// TIA Portal V17 export
// export: Created 2023-03-03T06:58:18.2471944Z, ExportSetting WithDefaults, DisplayName Totally Integrated Automation Portal, DisplayVersion V17 Update 5, DisplayName TIA Portal Openness, DisplayVersion V17 Update 5, DisplayName TIA Portal Version Control Interface, DisplayVersion V17, DisplayName SINAMICS Startdrive Advanced, DisplayVersion V17 SP1, DisplayName SINAMICS DCC, DisplayVersion V17 Update 1, DisplayName SINAMICS Startdrive G130, G150, S120, S150, SINAMICS MV, S210, DisplayVersion V17 SP1, DisplayName SINAMICS Startdrive G110M, G120, G120C, G120D, G120P, G115D, DisplayVersion V17 SP1, DisplayName STEP 7 Professional, DisplayVersion V17 Update 5, DisplayName STEP 7 Safety, DisplayVersion V17, DisplayName WinCC Advanced, DisplayVersion V17 Update 5
FUNCTION "Start motor HYD unit" : Void   // FC700, LAD
TITLE = FC Gestione accensione motori centralina HYD
{ S7_Optimized_Access := 'FALSE' }
AUTHOR : Max
FAMILY : Taglio
NAME : FC_START_MOTORI_CENTRALINA_HYD
VERSION : 0.1
// stored: AutoNumber false, IsIECCheckEnabled false, SetENOAutomatically false, UDAEnableTagReadback false
   VAR_TEMP
      cmd_Star : Bool;
      cmd_Triangle : Bool;
      cmd_recycling : Bool;
   END_VAR
   VAR_TEMP   // added for the SCL form of the ladder/FBD networks
      _w1 : Bool;
   END_VAR
BEGIN

REGION Network 1: *************************** Avviamento motore ricircolo **********************************
END_REGION

REGION Network 2: Condizioni per abilitazione avviamento motore ricircolo centralina
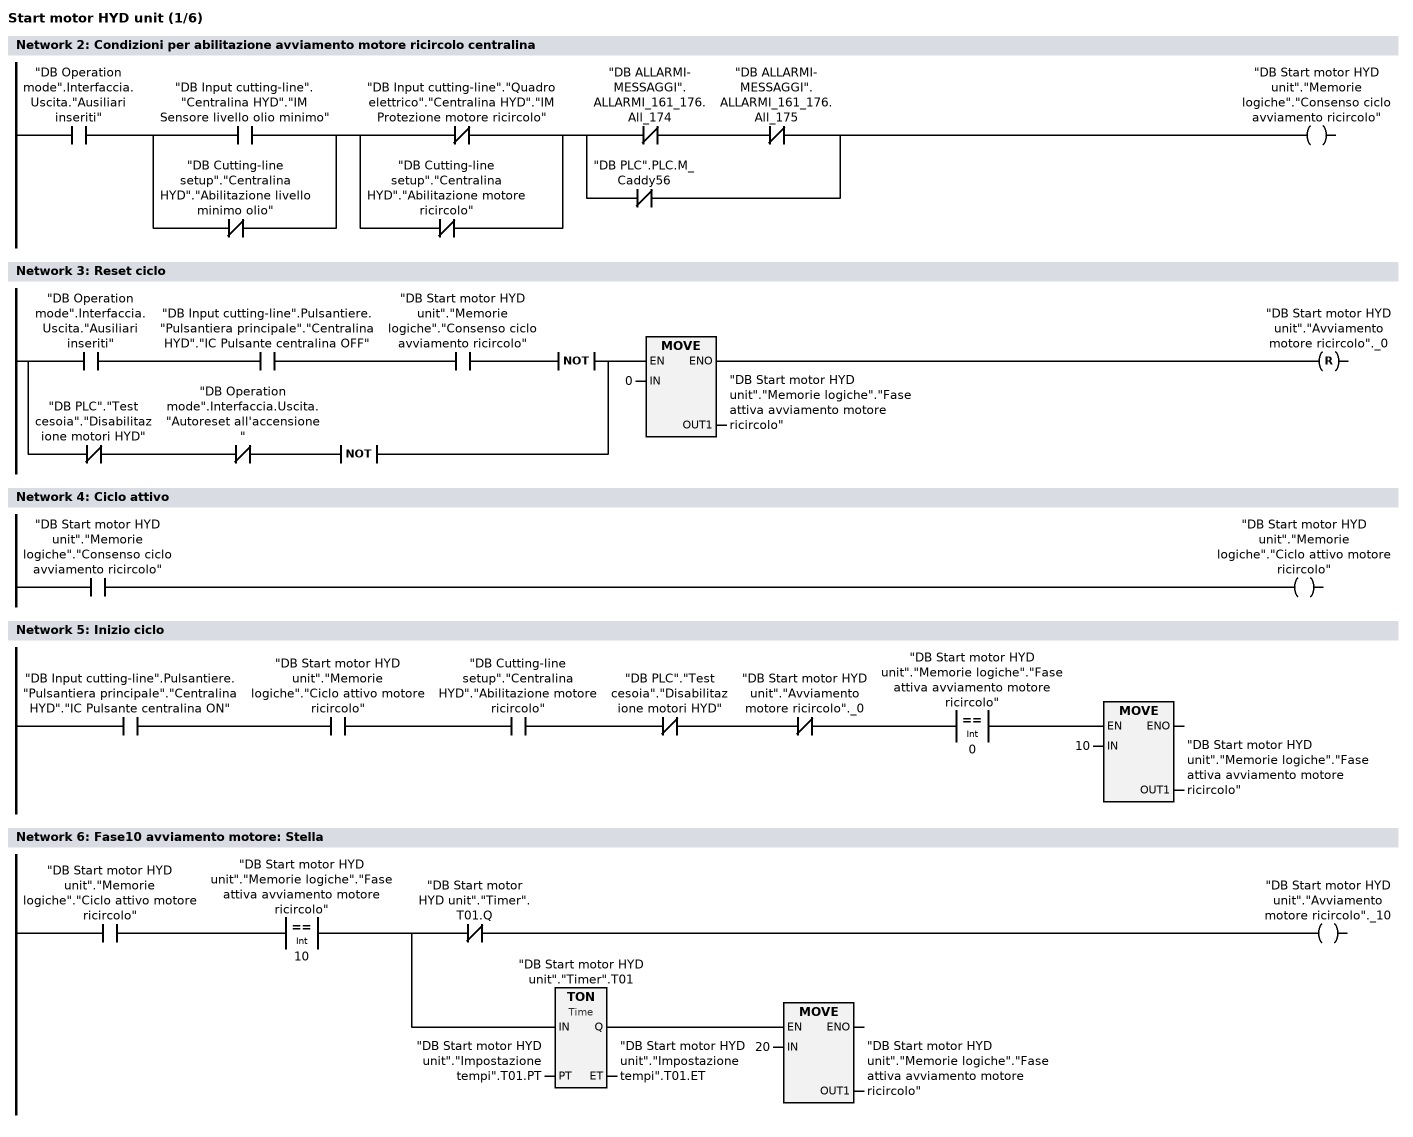
   RUNG wire#powerrail
      Contact( "DB Operation mode".Interfaccia.Uscita."Ausiliari inseriti" )
      wire#w1
      Contact( "DB Input cutting-line"."Centralina HYD"."IM Sensore livello olio minimo" )
      wire#w2
      I_Contact( "DB Input cutting-line"."Quadro elettrico"."Centralina HYD"."IM Protezione motore ricircolo" )
      wire#w3
      I_Contact( "DB ALLARMI-MESSAGGI".ALLARMI_161_176.All_174 )
      I_Contact( "DB ALLARMI-MESSAGGI".ALLARMI_161_176.All_175 )
      wire#w4
      Coil( "DB Start motor HYD unit"."Memorie logiche"."Consenso ciclo avviamento ricircolo" )
   END_RUNG
   RUNG wire#w1
      I_Contact( "DB Cutting-line setup"."Centralina HYD"."Abilitazione livello minimo olio" )
   END_RUNG wire#w2
   RUNG wire#w2
      I_Contact( "DB Cutting-line setup"."Centralina HYD"."Abilitazione motore ricircolo" )
   END_RUNG wire#w3
   RUNG wire#w3
      I_Contact( "DB PLC".PLC.M_Caddy56 )
   END_RUNG wire#w4
   // the same network as SCL:
   "DB Start motor HYD unit"."Memorie logiche"."Consenso ciclo avviamento ricircolo" := "DB Operation mode".Interfaccia.Uscita."Ausiliari inseriti" AND ("DB Input cutting-line"."Centralina HYD"."IM Sensore livello olio minimo" OR NOT "DB Cutting-line setup"."Centralina HYD"."Abilitazione livello minimo olio") AND (NOT "DB Input cutting-line"."Quadro elettrico"."Centralina HYD"."IM Protezione motore ricircolo" OR NOT "DB Cutting-line setup"."Centralina HYD"."Abilitazione motore ricircolo") AND ((NOT "DB ALLARMI-MESSAGGI".ALLARMI_161_176.All_174 AND NOT "DB ALLARMI-MESSAGGI".ALLARMI_161_176.All_175) OR NOT "DB PLC".PLC.M_Caddy56);
END_REGION

REGION Network 3: Reset ciclo
   RUNG wire#powerrail
      Contact( "DB Operation mode".Interfaccia.Uscita."Ausiliari inseriti" )
      Contact( "DB Input cutting-line".Pulsantiere."Pulsantiera principale"."Centralina HYD"."IC Pulsante centralina OFF" )
      Contact( "DB Start motor HYD unit"."Memorie logiche"."Consenso ciclo avviamento ricircolo" )
      Not()
      wire#w1
      Move(in := 0, out1 => "DB Start motor HYD unit"."Memorie logiche"."Fase attiva avviamento motore ricircolo")
      R_Coil( "DB Start motor HYD unit"."Avviamento motore ricircolo"._0 )
   END_RUNG
   RUNG wire#powerrail
      I_Contact( "DB PLC"."Test cesoia"."Disabilitazione motori HYD" )
      I_Contact( "DB Operation mode".Interfaccia.Uscita."Autoreset all'accensione" )
      Not()
   END_RUNG wire#w1
   // the same network as SCL:
   IF NOT ("DB Operation mode".Interfaccia.Uscita."Ausiliari inseriti" AND "DB Input cutting-line".Pulsantiere."Pulsantiera principale"."Centralina HYD"."IC Pulsante centralina OFF" AND "DB Start motor HYD unit"."Memorie logiche"."Consenso ciclo avviamento ricircolo") OR NOT (NOT "DB PLC"."Test cesoia"."Disabilitazione motori HYD" AND NOT "DB Operation mode".Interfaccia.Uscita."Autoreset all'accensione") THEN
       "DB Start motor HYD unit"."Memorie logiche"."Fase attiva avviamento motore ricircolo" := 0;
       "DB Start motor HYD unit"."Avviamento motore ricircolo"._0 := FALSE;
   END_IF;
END_REGION

REGION Network 4: Ciclo attivo
   RUNG wire#powerrail
      Contact( "DB Start motor HYD unit"."Memorie logiche"."Consenso ciclo avviamento ricircolo" )
      Coil( "DB Start motor HYD unit"."Memorie logiche"."Ciclo attivo motore ricircolo" )
   END_RUNG
   // the same network as SCL:
   "DB Start motor HYD unit"."Memorie logiche"."Ciclo attivo motore ricircolo" := "DB Start motor HYD unit"."Memorie logiche"."Consenso ciclo avviamento ricircolo";
END_REGION

REGION Network 5: Inizio ciclo
   RUNG wire#powerrail
      Contact( "DB Input cutting-line".Pulsantiere."Pulsantiera principale"."Centralina HYD"."IC Pulsante centralina ON" )
      Contact( "DB Start motor HYD unit"."Memorie logiche"."Ciclo attivo motore ricircolo" )
      Contact( "DB Cutting-line setup"."Centralina HYD"."Abilitazione motore ricircolo" )
      I_Contact( "DB PLC"."Test cesoia"."Disabilitazione motori HYD" )
      I_Contact( "DB Start motor HYD unit"."Avviamento motore ricircolo"._0 )
      { S7_Templates := "SrcType := Int" } EQ_Contact(in1 := "DB Start motor HYD unit"."Memorie logiche"."Fase attiva avviamento motore ricircolo", in2 := 0)
      Move(in := 10, out1 => "DB Start motor HYD unit"."Memorie logiche"."Fase attiva avviamento motore ricircolo")
   END_RUNG
   // the same network as SCL:
   IF "DB Input cutting-line".Pulsantiere."Pulsantiera principale"."Centralina HYD"."IC Pulsante centralina ON" AND "DB Start motor HYD unit"."Memorie logiche"."Ciclo attivo motore ricircolo" AND "DB Cutting-line setup"."Centralina HYD"."Abilitazione motore ricircolo" AND NOT "DB PLC"."Test cesoia"."Disabilitazione motori HYD" AND NOT "DB Start motor HYD unit"."Avviamento motore ricircolo"._0 AND ("DB Start motor HYD unit"."Memorie logiche"."Fase attiva avviamento motore ricircolo" = 0) THEN
       "DB Start motor HYD unit"."Memorie logiche"."Fase attiva avviamento motore ricircolo" := 10;
   END_IF;
END_REGION

REGION Network 6: Fase10 avviamento motore: Stella
   RUNG wire#powerrail
      Contact( "DB Start motor HYD unit"."Memorie logiche"."Ciclo attivo motore ricircolo" )
      { S7_Templates := "SrcType := Int" } EQ_Contact(in1 := "DB Start motor HYD unit"."Memorie logiche"."Fase attiva avviamento motore ricircolo", in2 := 10)
      wire#w1
      I_Contact( "DB Start motor HYD unit"."Timer".T01.Q )
      Coil( "DB Start motor HYD unit"."Avviamento motore ricircolo"._10 )
   END_RUNG
   RUNG wire#w1
      { S7_Templates := "time_type := Time" } "DB Start motor HYD unit"."Timer".T01.TON(pt := "DB Start motor HYD unit"."Impostazione tempi".T01.PT, et => "DB Start motor HYD unit"."Impostazione tempi".T01.ET)
      Move(in := 20, out1 => "DB Start motor HYD unit"."Memorie logiche"."Fase attiva avviamento motore ricircolo")
   END_RUNG
   // the same network as SCL:
   #_w1 := "DB Start motor HYD unit"."Memorie logiche"."Ciclo attivo motore ricircolo" AND ("DB Start motor HYD unit"."Memorie logiche"."Fase attiva avviamento motore ricircolo" = 10);
   "DB Start motor HYD unit"."Avviamento motore ricircolo"._10 := #_w1 AND NOT "DB Start motor HYD unit"."Timer".T01.Q;
   "DB Start motor HYD unit"."Timer".T01.TON(IN := #_w1,
                           PT := "DB Start motor HYD unit"."Impostazione tempi".T01.PT,
                           ET => "DB Start motor HYD unit"."Impostazione tempi".T01.ET);
   IF "DB Start motor HYD unit"."Timer".T01.Q THEN
       "DB Start motor HYD unit"."Memorie logiche"."Fase attiva avviamento motore ricircolo" := 20;
   END_IF;
END_REGION

REGION Network 7: Fase20 avviamento motore: Triangolo
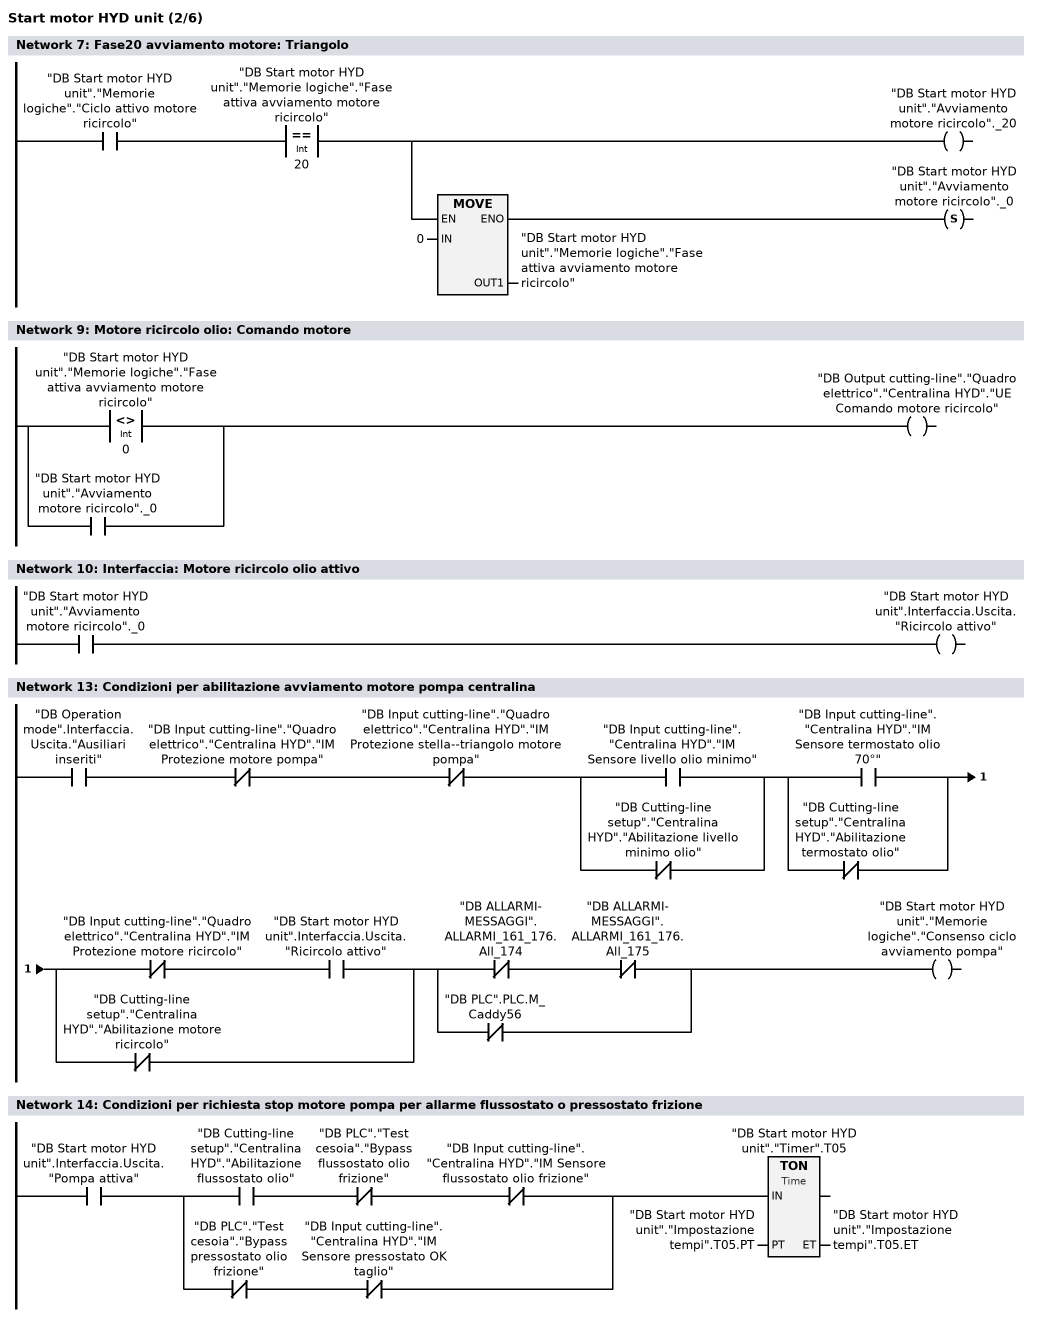
   RUNG wire#powerrail
      Contact( "DB Start motor HYD unit"."Memorie logiche"."Ciclo attivo motore ricircolo" )
      { S7_Templates := "SrcType := Int" } EQ_Contact(in1 := "DB Start motor HYD unit"."Memorie logiche"."Fase attiva avviamento motore ricircolo", in2 := 20)
      wire#w1
      Coil( "DB Start motor HYD unit"."Avviamento motore ricircolo"._20 )
   END_RUNG
   RUNG wire#w1
      Move(in := 0, out1 => "DB Start motor HYD unit"."Memorie logiche"."Fase attiva avviamento motore ricircolo")
      S_Coil( "DB Start motor HYD unit"."Avviamento motore ricircolo"._0 )
   END_RUNG
   // the same network as SCL:
   "DB Start motor HYD unit"."Avviamento motore ricircolo"._20 := "DB Start motor HYD unit"."Memorie logiche"."Ciclo attivo motore ricircolo" AND ("DB Start motor HYD unit"."Memorie logiche"."Fase attiva avviamento motore ricircolo" = 20);
   IF "DB Start motor HYD unit"."Avviamento motore ricircolo"._20 THEN
       "DB Start motor HYD unit"."Memorie logiche"."Fase attiva avviamento motore ricircolo" := 0;
       "DB Start motor HYD unit"."Avviamento motore ricircolo"._0 := TRUE;
   END_IF;
END_REGION

REGION Network 8: Dummy
END_REGION

REGION Network 9: Motore ricircolo olio: Comando motore
   RUNG wire#powerrail
      { S7_Templates := "SrcType := Int" } NE_Contact(in1 := "DB Start motor HYD unit"."Memorie logiche"."Fase attiva avviamento motore ricircolo", in2 := 0)
      wire#w1
      Coil( "DB Output cutting-line"."Quadro elettrico"."Centralina HYD"."UE Comando motore ricircolo" )
   END_RUNG
   RUNG wire#powerrail
      Contact( "DB Start motor HYD unit"."Avviamento motore ricircolo"._0 )
   END_RUNG wire#w1
   // the same network as SCL:
   "DB Output cutting-line"."Quadro elettrico"."Centralina HYD"."UE Comando motore ricircolo" := ("DB Start motor HYD unit"."Memorie logiche"."Fase attiva avviamento motore ricircolo" <> 0) OR "DB Start motor HYD unit"."Avviamento motore ricircolo"._0;
END_REGION

REGION Network 10: Interfaccia: Motore ricircolo olio attivo
   RUNG wire#powerrail
      Contact( "DB Start motor HYD unit"."Avviamento motore ricircolo"._0 )
      Coil( "DB Start motor HYD unit".Interfaccia.Uscita."Ricircolo attivo" )
   END_RUNG
   // the same network as SCL:
   "DB Start motor HYD unit".Interfaccia.Uscita."Ricircolo attivo" := "DB Start motor HYD unit"."Avviamento motore ricircolo"._0;
END_REGION

REGION Network 11: Dummy
END_REGION

REGION Network 12: *********************** Avviamento motore pompa principale ******************************
END_REGION

REGION Network 13: Condizioni per abilitazione avviamento motore pompa centralina
   RUNG wire#powerrail
      Contact( "DB Operation mode".Interfaccia.Uscita."Ausiliari inseriti" )
      I_Contact( "DB Input cutting-line"."Quadro elettrico"."Centralina HYD"."IM Protezione motore pompa" )
      I_Contact( "DB Input cutting-line"."Quadro elettrico"."Centralina HYD"."IM Protezione stella--triangolo motore pompa" )
      wire#w1
      Contact( "DB Input cutting-line"."Centralina HYD"."IM Sensore livello olio minimo" )
      wire#w2
      Contact( "DB Input cutting-line"."Centralina HYD"."IM Sensore termostato olio 70°" )
      wire#w3
      I_Contact( "DB Input cutting-line"."Quadro elettrico"."Centralina HYD"."IM Protezione motore ricircolo" )
      Contact( "DB Start motor HYD unit".Interfaccia.Uscita."Ricircolo attivo" )
      wire#w4
      I_Contact( "DB ALLARMI-MESSAGGI".ALLARMI_161_176.All_174 )
      I_Contact( "DB ALLARMI-MESSAGGI".ALLARMI_161_176.All_175 )
      wire#w5
      Coil( "DB Start motor HYD unit"."Memorie logiche"."Consenso ciclo avviamento pompa" )
   END_RUNG
   RUNG wire#w1
      I_Contact( "DB Cutting-line setup"."Centralina HYD"."Abilitazione livello minimo olio" )
   END_RUNG wire#w2
   RUNG wire#w2
      I_Contact( "DB Cutting-line setup"."Centralina HYD"."Abilitazione termostato olio" )
   END_RUNG wire#w3
   RUNG wire#w3
      I_Contact( "DB Cutting-line setup"."Centralina HYD"."Abilitazione motore ricircolo" )
   END_RUNG wire#w4
   RUNG wire#w4
      I_Contact( "DB PLC".PLC.M_Caddy56 )
   END_RUNG wire#w5
   // the same network as SCL:
   "DB Start motor HYD unit"."Memorie logiche"."Consenso ciclo avviamento pompa" := "DB Operation mode".Interfaccia.Uscita."Ausiliari inseriti" AND NOT "DB Input cutting-line"."Quadro elettrico"."Centralina HYD"."IM Protezione motore pompa" AND NOT "DB Input cutting-line"."Quadro elettrico"."Centralina HYD"."IM Protezione stella--triangolo motore pompa" AND ("DB Input cutting-line"."Centralina HYD"."IM Sensore livello olio minimo" OR NOT "DB Cutting-line setup"."Centralina HYD"."Abilitazione livello minimo olio") AND ("DB Input cutting-line"."Centralina HYD"."IM Sensore termostato olio 70°" OR NOT "DB Cutting-line setup"."Centralina HYD"."Abilitazione termostato olio") AND ((NOT "DB Input cutting-line"."Quadro elettrico"."Centralina HYD"."IM Protezione motore ricircolo" AND "DB Start motor HYD unit".Interfaccia.Uscita."Ricircolo attivo") OR NOT "DB Cutting-line setup"."Centralina HYD"."Abilitazione motore ricircolo") AND ((NOT "DB ALLARMI-MESSAGGI".ALLARMI_161_176.All_174 AND NOT "DB ALLARMI-MESSAGGI".ALLARMI_161_176.All_175) OR NOT "DB PLC".PLC.M_Caddy56);
END_REGION

REGION Network 14: Condizioni per richiesta stop motore pompa per allarme flussostato o pressostato frizione
   RUNG wire#powerrail
      Contact( "DB Start motor HYD unit".Interfaccia.Uscita."Pompa attiva" )
      wire#w1
      Contact( "DB Cutting-line setup"."Centralina HYD"."Abilitazione flussostato olio" )
      I_Contact( "DB PLC"."Test cesoia"."Bypass flussostato olio frizione" )
      I_Contact( "DB Input cutting-line"."Centralina HYD"."IM Sensore flussostato olio frizione" )
      wire#w2
      { S7_Templates := "time_type := Time" } "DB Start motor HYD unit"."Timer".T05.TON(pt := "DB Start motor HYD unit"."Impostazione tempi".T05.PT, et => "DB Start motor HYD unit"."Impostazione tempi".T05.ET)
   END_RUNG
   RUNG wire#w1
      I_Contact( "DB PLC"."Test cesoia"."Bypass pressostato olio frizione" )
      I_Contact( "DB Input cutting-line"."Centralina HYD"."IM Sensore pressostato OK taglio" )
   END_RUNG wire#w2
   // the same network as SCL:
   "DB Start motor HYD unit"."Timer".T05.TON(IN := "DB Start motor HYD unit".Interfaccia.Uscita."Pompa attiva" AND (("DB Cutting-line setup"."Centralina HYD"."Abilitazione flussostato olio" AND NOT "DB PLC"."Test cesoia"."Bypass flussostato olio frizione" AND NOT "DB Input cutting-line"."Centralina HYD"."IM Sensore flussostato olio frizione") OR (NOT "DB PLC"."Test cesoia"."Bypass pressostato olio frizione" AND NOT "DB Input cutting-line"."Centralina HYD"."IM Sensore pressostato OK taglio")),
                           PT := "DB Start motor HYD unit"."Impostazione tempi".T05.PT,
                           ET => "DB Start motor HYD unit"."Impostazione tempi".T05.ET);
END_REGION

REGION Network 15: Richiesta stop motore pompa per allarmi
   // Nel caso in cui avvengano allarmi viene usata questa richiesta. Cmq allo spegnimento degli ausiliari la pompa viene fermata dalla memoria "Ausiliari inseriti"
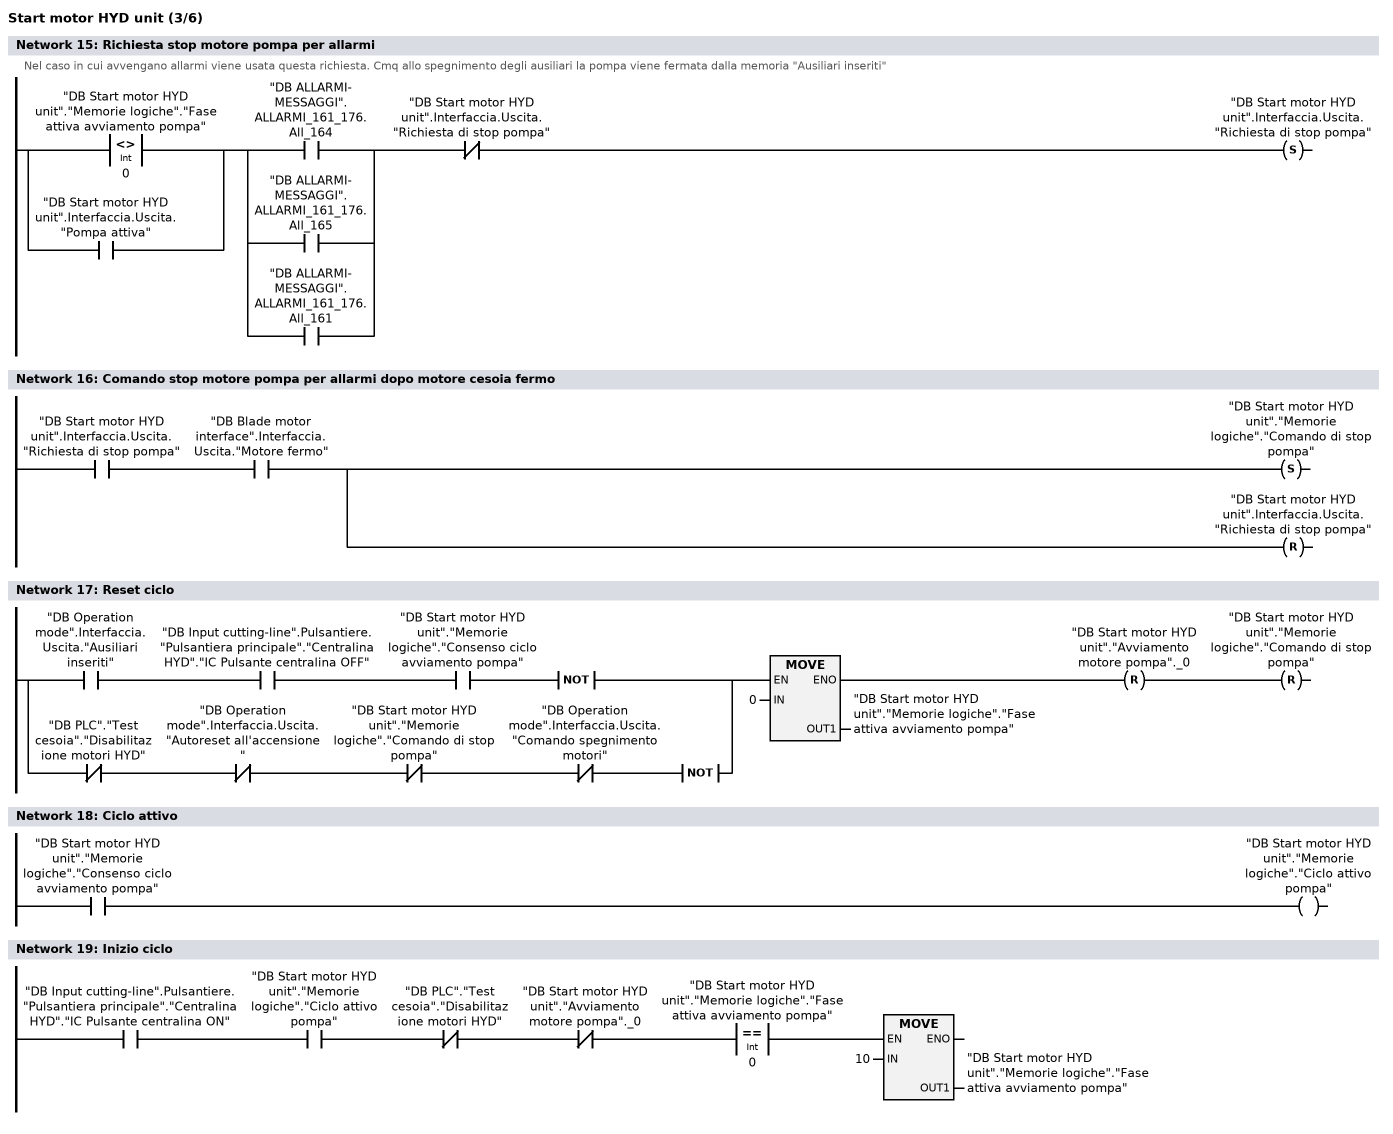
   RUNG wire#powerrail
      { S7_Templates := "SrcType := Int" } NE_Contact(in1 := "DB Start motor HYD unit"."Memorie logiche"."Fase attiva avviamento pompa", in2 := 0)
      wire#w1
      Contact( "DB ALLARMI-MESSAGGI".ALLARMI_161_176.All_164 )
      wire#w2
      I_Contact( "DB Start motor HYD unit".Interfaccia.Uscita."Richiesta di stop pompa" )
      S_Coil( "DB Start motor HYD unit".Interfaccia.Uscita."Richiesta di stop pompa" )
   END_RUNG
   RUNG wire#powerrail
      Contact( "DB Start motor HYD unit".Interfaccia.Uscita."Pompa attiva" )
   END_RUNG wire#w1
   RUNG wire#w1
      Contact( "DB ALLARMI-MESSAGGI".ALLARMI_161_176.All_165 )
   END_RUNG wire#w2
   RUNG wire#w1
      Contact( "DB ALLARMI-MESSAGGI".ALLARMI_161_176.All_161 )
   END_RUNG wire#w2
   // the same network as SCL:
   IF (("DB Start motor HYD unit"."Memorie logiche"."Fase attiva avviamento pompa" <> 0) OR "DB Start motor HYD unit".Interfaccia.Uscita."Pompa attiva") AND ("DB ALLARMI-MESSAGGI".ALLARMI_161_176.All_164 OR "DB ALLARMI-MESSAGGI".ALLARMI_161_176.All_165 OR "DB ALLARMI-MESSAGGI".ALLARMI_161_176.All_161) AND NOT "DB Start motor HYD unit".Interfaccia.Uscita."Richiesta di stop pompa" THEN
       "DB Start motor HYD unit".Interfaccia.Uscita."Richiesta di stop pompa" := TRUE;
   END_IF;
END_REGION

REGION Network 16: Comando stop motore pompa per allarmi dopo motore cesoia fermo
   RUNG wire#powerrail
      Contact( "DB Start motor HYD unit".Interfaccia.Uscita."Richiesta di stop pompa" )
      Contact( "DB Blade motor interface".Interfaccia.Uscita."Motore fermo" )
      wire#w1
      S_Coil( "DB Start motor HYD unit"."Memorie logiche"."Comando di stop pompa" )
   END_RUNG
   RUNG wire#w1
      R_Coil( "DB Start motor HYD unit".Interfaccia.Uscita."Richiesta di stop pompa" )
   END_RUNG
   // the same network as SCL:
   IF "DB Start motor HYD unit".Interfaccia.Uscita."Richiesta di stop pompa" AND "DB Blade motor interface".Interfaccia.Uscita."Motore fermo" THEN
       "DB Start motor HYD unit"."Memorie logiche"."Comando di stop pompa" := TRUE;
       "DB Start motor HYD unit".Interfaccia.Uscita."Richiesta di stop pompa" := FALSE;
   END_IF;
END_REGION

REGION Network 17: Reset ciclo
   RUNG wire#powerrail
      Contact( "DB Operation mode".Interfaccia.Uscita."Ausiliari inseriti" )
      Contact( "DB Input cutting-line".Pulsantiere."Pulsantiera principale"."Centralina HYD"."IC Pulsante centralina OFF" )
      Contact( "DB Start motor HYD unit"."Memorie logiche"."Consenso ciclo avviamento pompa" )
      Not()
      wire#w1
      Move(in := 0, out1 => "DB Start motor HYD unit"."Memorie logiche"."Fase attiva avviamento pompa")
      R_Coil( "DB Start motor HYD unit"."Avviamento motore pompa"._0 )
      R_Coil( "DB Start motor HYD unit"."Memorie logiche"."Comando di stop pompa" )
   END_RUNG
   RUNG wire#powerrail
      I_Contact( "DB PLC"."Test cesoia"."Disabilitazione motori HYD" )
      I_Contact( "DB Operation mode".Interfaccia.Uscita."Autoreset all'accensione" )
      I_Contact( "DB Start motor HYD unit"."Memorie logiche"."Comando di stop pompa" )
      I_Contact( "DB Operation mode".Interfaccia.Uscita."Comando spegnimento motori" )
      Not()
   END_RUNG wire#w1
   // the same network as SCL:
   IF NOT ("DB Operation mode".Interfaccia.Uscita."Ausiliari inseriti" AND "DB Input cutting-line".Pulsantiere."Pulsantiera principale"."Centralina HYD"."IC Pulsante centralina OFF" AND "DB Start motor HYD unit"."Memorie logiche"."Consenso ciclo avviamento pompa") OR NOT (NOT "DB PLC"."Test cesoia"."Disabilitazione motori HYD" AND NOT "DB Operation mode".Interfaccia.Uscita."Autoreset all'accensione" AND NOT "DB Start motor HYD unit"."Memorie logiche"."Comando di stop pompa" AND NOT "DB Operation mode".Interfaccia.Uscita."Comando spegnimento motori") THEN
       "DB Start motor HYD unit"."Memorie logiche"."Fase attiva avviamento pompa" := 0;
       "DB Start motor HYD unit"."Avviamento motore pompa"._0 := FALSE;
       "DB Start motor HYD unit"."Memorie logiche"."Comando di stop pompa" := FALSE;
   END_IF;
END_REGION

REGION Network 18: Ciclo attivo
   RUNG wire#powerrail
      Contact( "DB Start motor HYD unit"."Memorie logiche"."Consenso ciclo avviamento pompa" )
      Coil( "DB Start motor HYD unit"."Memorie logiche"."Ciclo attivo pompa" )
   END_RUNG
   // the same network as SCL:
   "DB Start motor HYD unit"."Memorie logiche"."Ciclo attivo pompa" := "DB Start motor HYD unit"."Memorie logiche"."Consenso ciclo avviamento pompa";
END_REGION

REGION Network 19: Inizio ciclo
   RUNG wire#powerrail
      Contact( "DB Input cutting-line".Pulsantiere."Pulsantiera principale"."Centralina HYD"."IC Pulsante centralina ON" )
      Contact( "DB Start motor HYD unit"."Memorie logiche"."Ciclo attivo pompa" )
      I_Contact( "DB PLC"."Test cesoia"."Disabilitazione motori HYD" )
      I_Contact( "DB Start motor HYD unit"."Avviamento motore pompa"._0 )
      { S7_Templates := "SrcType := Int" } EQ_Contact(in1 := "DB Start motor HYD unit"."Memorie logiche"."Fase attiva avviamento pompa", in2 := 0)
      Move(in := 10, out1 => "DB Start motor HYD unit"."Memorie logiche"."Fase attiva avviamento pompa")
   END_RUNG
   // the same network as SCL:
   IF "DB Input cutting-line".Pulsantiere."Pulsantiera principale"."Centralina HYD"."IC Pulsante centralina ON" AND "DB Start motor HYD unit"."Memorie logiche"."Ciclo attivo pompa" AND NOT "DB PLC"."Test cesoia"."Disabilitazione motori HYD" AND NOT "DB Start motor HYD unit"."Avviamento motore pompa"._0 AND ("DB Start motor HYD unit"."Memorie logiche"."Fase attiva avviamento pompa" = 0) THEN
       "DB Start motor HYD unit"."Memorie logiche"."Fase attiva avviamento pompa" := 10;
   END_IF;
END_REGION

REGION Network 20: Fase10 avviamento motore: Stella
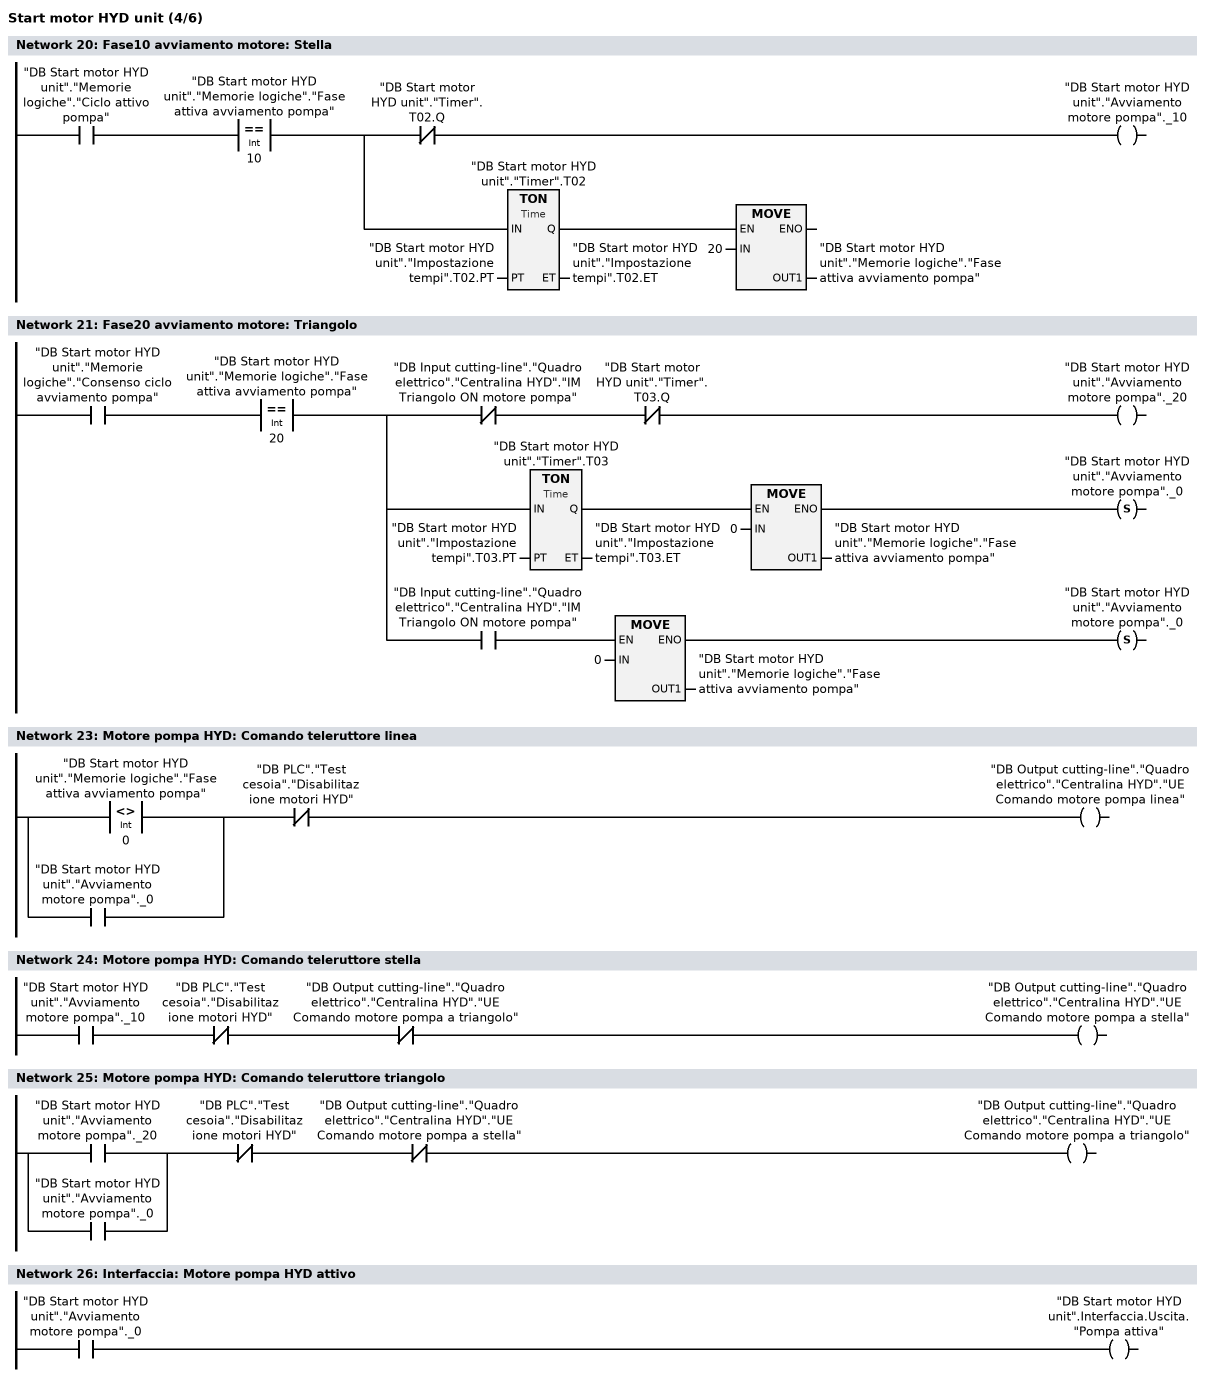
   RUNG wire#powerrail
      Contact( "DB Start motor HYD unit"."Memorie logiche"."Ciclo attivo pompa" )
      { S7_Templates := "SrcType := Int" } EQ_Contact(in1 := "DB Start motor HYD unit"."Memorie logiche"."Fase attiva avviamento pompa", in2 := 10)
      wire#w1
      I_Contact( "DB Start motor HYD unit"."Timer".T02.Q )
      Coil( "DB Start motor HYD unit"."Avviamento motore pompa"._10 )
   END_RUNG
   RUNG wire#w1
      { S7_Templates := "time_type := Time" } "DB Start motor HYD unit"."Timer".T02.TON(pt := "DB Start motor HYD unit"."Impostazione tempi".T02.PT, et => "DB Start motor HYD unit"."Impostazione tempi".T02.ET)
      Move(in := 20, out1 => "DB Start motor HYD unit"."Memorie logiche"."Fase attiva avviamento pompa")
   END_RUNG
   // the same network as SCL:
   #_w1 := "DB Start motor HYD unit"."Memorie logiche"."Ciclo attivo pompa" AND ("DB Start motor HYD unit"."Memorie logiche"."Fase attiva avviamento pompa" = 10);
   "DB Start motor HYD unit"."Avviamento motore pompa"._10 := #_w1 AND NOT "DB Start motor HYD unit"."Timer".T02.Q;
   "DB Start motor HYD unit"."Timer".T02.TON(IN := #_w1,
                           PT := "DB Start motor HYD unit"."Impostazione tempi".T02.PT,
                           ET => "DB Start motor HYD unit"."Impostazione tempi".T02.ET);
   IF "DB Start motor HYD unit"."Timer".T02.Q THEN
       "DB Start motor HYD unit"."Memorie logiche"."Fase attiva avviamento pompa" := 20;
   END_IF;
END_REGION

REGION Network 21: Fase20 avviamento motore: Triangolo
   RUNG wire#powerrail
      Contact( "DB Start motor HYD unit"."Memorie logiche"."Consenso ciclo avviamento pompa" )
      { S7_Templates := "SrcType := Int" } EQ_Contact(in1 := "DB Start motor HYD unit"."Memorie logiche"."Fase attiva avviamento pompa", in2 := 20)
      wire#w1
      I_Contact( "DB Input cutting-line"."Quadro elettrico"."Centralina HYD"."IM Triangolo ON motore pompa" )
      I_Contact( "DB Start motor HYD unit"."Timer".T03.Q )
      Coil( "DB Start motor HYD unit"."Avviamento motore pompa"._20 )
   END_RUNG
   RUNG wire#w1
      { S7_Templates := "time_type := Time" } "DB Start motor HYD unit"."Timer".T03.TON(pt := "DB Start motor HYD unit"."Impostazione tempi".T03.PT, et => "DB Start motor HYD unit"."Impostazione tempi".T03.ET)
      Move(in := 0, out1 => "DB Start motor HYD unit"."Memorie logiche"."Fase attiva avviamento pompa")
      S_Coil( "DB Start motor HYD unit"."Avviamento motore pompa"._0 )
   END_RUNG
   RUNG wire#w1
      Contact( "DB Input cutting-line"."Quadro elettrico"."Centralina HYD"."IM Triangolo ON motore pompa" )
      Move(in := 0, out1 => "DB Start motor HYD unit"."Memorie logiche"."Fase attiva avviamento pompa")
      S_Coil( "DB Start motor HYD unit"."Avviamento motore pompa"._0 )
   END_RUNG
   // the same network as SCL:
   #_w1 := "DB Start motor HYD unit"."Memorie logiche"."Consenso ciclo avviamento pompa" AND ("DB Start motor HYD unit"."Memorie logiche"."Fase attiva avviamento pompa" = 20);
   "DB Start motor HYD unit"."Avviamento motore pompa"._20 := #_w1 AND NOT "DB Input cutting-line"."Quadro elettrico"."Centralina HYD"."IM Triangolo ON motore pompa" AND NOT "DB Start motor HYD unit"."Timer".T03.Q;
   "DB Start motor HYD unit"."Timer".T03.TON(IN := #_w1,
                           PT := "DB Start motor HYD unit"."Impostazione tempi".T03.PT,
                           ET => "DB Start motor HYD unit"."Impostazione tempi".T03.ET);
   IF "DB Start motor HYD unit"."Timer".T03.Q THEN
       "DB Start motor HYD unit"."Memorie logiche"."Fase attiva avviamento pompa" := 0;
       "DB Start motor HYD unit"."Avviamento motore pompa"._0 := TRUE;
   END_IF;
   IF #_w1 AND "DB Input cutting-line"."Quadro elettrico"."Centralina HYD"."IM Triangolo ON motore pompa" THEN
       "DB Start motor HYD unit"."Memorie logiche"."Fase attiva avviamento pompa" := 0;
       "DB Start motor HYD unit"."Avviamento motore pompa"._0 := TRUE;
   END_IF;
END_REGION

REGION Network 22: Dummy
END_REGION

REGION Network 23: Motore pompa HYD: Comando teleruttore linea
   RUNG wire#powerrail
      { S7_Templates := "SrcType := Int" } NE_Contact(in1 := "DB Start motor HYD unit"."Memorie logiche"."Fase attiva avviamento pompa", in2 := 0)
      wire#w1
      I_Contact( "DB PLC"."Test cesoia"."Disabilitazione motori HYD" )
      Coil( "DB Output cutting-line"."Quadro elettrico"."Centralina HYD"."UE Comando motore pompa linea" )
   END_RUNG
   RUNG wire#powerrail
      Contact( "DB Start motor HYD unit"."Avviamento motore pompa"._0 )
   END_RUNG wire#w1
   // the same network as SCL:
   "DB Output cutting-line"."Quadro elettrico"."Centralina HYD"."UE Comando motore pompa linea" := (("DB Start motor HYD unit"."Memorie logiche"."Fase attiva avviamento pompa" <> 0) OR "DB Start motor HYD unit"."Avviamento motore pompa"._0) AND NOT "DB PLC"."Test cesoia"."Disabilitazione motori HYD";
END_REGION

REGION Network 24: Motore pompa HYD: Comando teleruttore stella
   RUNG wire#powerrail
      Contact( "DB Start motor HYD unit"."Avviamento motore pompa"._10 )
      I_Contact( "DB PLC"."Test cesoia"."Disabilitazione motori HYD" )
      I_Contact( "DB Output cutting-line"."Quadro elettrico"."Centralina HYD"."UE Comando motore pompa a triangolo" )
      Coil( "DB Output cutting-line"."Quadro elettrico"."Centralina HYD"."UE Comando motore pompa a stella" )
   END_RUNG
   // the same network as SCL:
   "DB Output cutting-line"."Quadro elettrico"."Centralina HYD"."UE Comando motore pompa a stella" := "DB Start motor HYD unit"."Avviamento motore pompa"._10 AND NOT "DB PLC"."Test cesoia"."Disabilitazione motori HYD" AND NOT "DB Output cutting-line"."Quadro elettrico"."Centralina HYD"."UE Comando motore pompa a triangolo";
END_REGION

REGION Network 25: Motore pompa HYD: Comando teleruttore triangolo
   RUNG wire#powerrail
      Contact( "DB Start motor HYD unit"."Avviamento motore pompa"._20 )
      wire#w1
      I_Contact( "DB PLC"."Test cesoia"."Disabilitazione motori HYD" )
      I_Contact( "DB Output cutting-line"."Quadro elettrico"."Centralina HYD"."UE Comando motore pompa a stella" )
      Coil( "DB Output cutting-line"."Quadro elettrico"."Centralina HYD"."UE Comando motore pompa a triangolo" )
   END_RUNG
   RUNG wire#powerrail
      Contact( "DB Start motor HYD unit"."Avviamento motore pompa"._0 )
   END_RUNG wire#w1
   // the same network as SCL:
   "DB Output cutting-line"."Quadro elettrico"."Centralina HYD"."UE Comando motore pompa a triangolo" := ("DB Start motor HYD unit"."Avviamento motore pompa"._20 OR "DB Start motor HYD unit"."Avviamento motore pompa"._0) AND NOT "DB PLC"."Test cesoia"."Disabilitazione motori HYD" AND NOT "DB Output cutting-line"."Quadro elettrico"."Centralina HYD"."UE Comando motore pompa a stella";
END_REGION

REGION Network 26: Interfaccia: Motore pompa HYD attivo
   RUNG wire#powerrail
      Contact( "DB Start motor HYD unit"."Avviamento motore pompa"._0 )
      Coil( "DB Start motor HYD unit".Interfaccia.Uscita."Pompa attiva" )
   END_RUNG
   // the same network as SCL:
   "DB Start motor HYD unit".Interfaccia.Uscita."Pompa attiva" := "DB Start motor HYD unit"."Avviamento motore pompa"._0;
END_REGION

REGION Network 27: Dummy
END_REGION

REGION Network 28: Comando valvola pressione olio cesoia
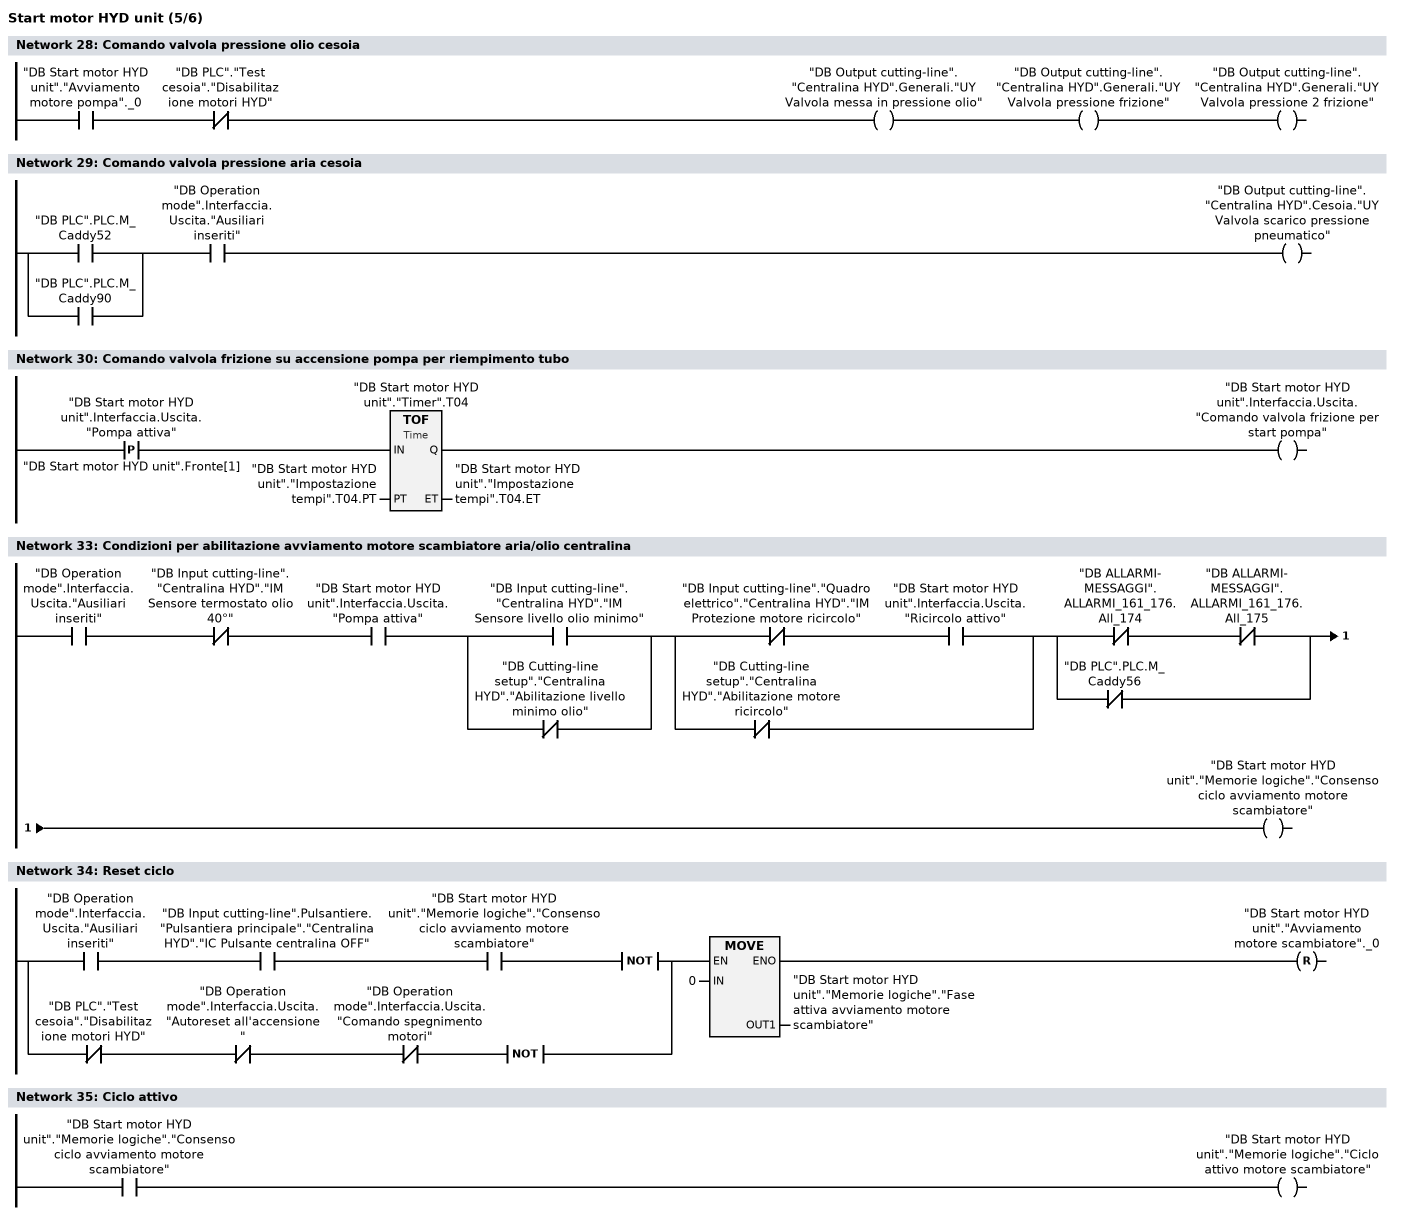
   RUNG wire#powerrail
      Contact( "DB Start motor HYD unit"."Avviamento motore pompa"._0 )
      I_Contact( "DB PLC"."Test cesoia"."Disabilitazione motori HYD" )
      Coil( "DB Output cutting-line"."Centralina HYD".Generali."UY Valvola messa in pressione olio" )
      Coil( "DB Output cutting-line"."Centralina HYD".Generali."UY Valvola pressione frizione" )
      Coil( "DB Output cutting-line"."Centralina HYD".Generali."UY Valvola pressione 2 frizione" )
   END_RUNG
   // the same network as SCL:
   "DB Output cutting-line"."Centralina HYD".Generali."UY Valvola messa in pressione olio" := "DB Start motor HYD unit"."Avviamento motore pompa"._0 AND NOT "DB PLC"."Test cesoia"."Disabilitazione motori HYD";
   "DB Output cutting-line"."Centralina HYD".Generali."UY Valvola pressione frizione" := "DB Output cutting-line"."Centralina HYD".Generali."UY Valvola messa in pressione olio";
   "DB Output cutting-line"."Centralina HYD".Generali."UY Valvola pressione 2 frizione" := "DB Output cutting-line"."Centralina HYD".Generali."UY Valvola messa in pressione olio";
END_REGION

REGION Network 29: Comando valvola pressione aria cesoia
   RUNG wire#powerrail
      Contact( "DB PLC".PLC.M_Caddy52 )
      wire#w1
      Contact( "DB Operation mode".Interfaccia.Uscita."Ausiliari inseriti" )
      Coil( "DB Output cutting-line"."Centralina HYD".Cesoia."UY Valvola scarico pressione pneumatico" )
   END_RUNG
   RUNG wire#powerrail
      Contact( "DB PLC".PLC.M_Caddy90 )
   END_RUNG wire#w1
   // the same network as SCL:
   "DB Output cutting-line"."Centralina HYD".Cesoia."UY Valvola scarico pressione pneumatico" := ("DB PLC".PLC.M_Caddy52 OR "DB PLC".PLC.M_Caddy90) AND "DB Operation mode".Interfaccia.Uscita."Ausiliari inseriti";
END_REGION

REGION Network 30: Comando valvola frizione su accensione pompa per riempimento tubo
   RUNG wire#powerrail
      P_Contact(operand := "DB Start motor HYD unit".Interfaccia.Uscita."Pompa attiva", bit := "DB Start motor HYD unit".Fronte[1])
      { S7_Templates := "time_type := Time" } "DB Start motor HYD unit"."Timer".T04.TOF(pt := "DB Start motor HYD unit"."Impostazione tempi".T04.PT, et => "DB Start motor HYD unit"."Impostazione tempi".T04.ET)
      Coil( "DB Start motor HYD unit".Interfaccia.Uscita."Comando valvola frizione per start pompa" )
   END_RUNG
   // the same network as SCL:
   #_w1 := "DB Start motor HYD unit".Interfaccia.Uscita."Pompa attiva" AND NOT "DB Start motor HYD unit".Fronte[1];   // rising edge of "DB Start motor HYD unit".Interfaccia.Uscita."Pompa attiva"
   "DB Start motor HYD unit".Fronte[1] := "DB Start motor HYD unit".Interfaccia.Uscita."Pompa attiva";
   "DB Start motor HYD unit"."Timer".T04.TOF(IN := #_w1,
                           PT := "DB Start motor HYD unit"."Impostazione tempi".T04.PT,
                           ET => "DB Start motor HYD unit"."Impostazione tempi".T04.ET);
   "DB Start motor HYD unit".Interfaccia.Uscita."Comando valvola frizione per start pompa" := "DB Start motor HYD unit"."Timer".T04.Q;
END_REGION

REGION Network 31: Dummy
END_REGION

REGION Network 32: *********************** Avviamento motore scambiatore aria/olio ****************************
END_REGION

REGION Network 33: Condizioni per abilitazione avviamento motore scambiatore aria/olio centralina
   RUNG wire#powerrail
      Contact( "DB Operation mode".Interfaccia.Uscita."Ausiliari inseriti" )
      I_Contact( "DB Input cutting-line"."Centralina HYD"."IM Sensore termostato olio 40°" )
      Contact( "DB Start motor HYD unit".Interfaccia.Uscita."Pompa attiva" )
      wire#w1
      Contact( "DB Input cutting-line"."Centralina HYD"."IM Sensore livello olio minimo" )
      wire#w2
      I_Contact( "DB Input cutting-line"."Quadro elettrico"."Centralina HYD"."IM Protezione motore ricircolo" )
      Contact( "DB Start motor HYD unit".Interfaccia.Uscita."Ricircolo attivo" )
      wire#w3
      I_Contact( "DB ALLARMI-MESSAGGI".ALLARMI_161_176.All_174 )
      I_Contact( "DB ALLARMI-MESSAGGI".ALLARMI_161_176.All_175 )
      wire#w4
      Coil( "DB Start motor HYD unit"."Memorie logiche"."Consenso ciclo avviamento motore scambiatore" )
   END_RUNG
   RUNG wire#w1
      I_Contact( "DB Cutting-line setup"."Centralina HYD"."Abilitazione livello minimo olio" )
   END_RUNG wire#w2
   RUNG wire#w2
      I_Contact( "DB Cutting-line setup"."Centralina HYD"."Abilitazione motore ricircolo" )
   END_RUNG wire#w3
   RUNG wire#w3
      I_Contact( "DB PLC".PLC.M_Caddy56 )
   END_RUNG wire#w4
   // the same network as SCL:
   "DB Start motor HYD unit"."Memorie logiche"."Consenso ciclo avviamento motore scambiatore" := "DB Operation mode".Interfaccia.Uscita."Ausiliari inseriti" AND NOT "DB Input cutting-line"."Centralina HYD"."IM Sensore termostato olio 40°" AND "DB Start motor HYD unit".Interfaccia.Uscita."Pompa attiva" AND ("DB Input cutting-line"."Centralina HYD"."IM Sensore livello olio minimo" OR NOT "DB Cutting-line setup"."Centralina HYD"."Abilitazione livello minimo olio") AND ((NOT "DB Input cutting-line"."Quadro elettrico"."Centralina HYD"."IM Protezione motore ricircolo" AND "DB Start motor HYD unit".Interfaccia.Uscita."Ricircolo attivo") OR NOT "DB Cutting-line setup"."Centralina HYD"."Abilitazione motore ricircolo") AND ((NOT "DB ALLARMI-MESSAGGI".ALLARMI_161_176.All_174 AND NOT "DB ALLARMI-MESSAGGI".ALLARMI_161_176.All_175) OR NOT "DB PLC".PLC.M_Caddy56);
END_REGION

REGION Network 34: Reset ciclo
   RUNG wire#powerrail
      Contact( "DB Operation mode".Interfaccia.Uscita."Ausiliari inseriti" )
      Contact( "DB Input cutting-line".Pulsantiere."Pulsantiera principale"."Centralina HYD"."IC Pulsante centralina OFF" )
      Contact( "DB Start motor HYD unit"."Memorie logiche"."Consenso ciclo avviamento motore scambiatore" )
      Not()
      wire#w1
      Move(in := 0, out1 => "DB Start motor HYD unit"."Memorie logiche"."Fase attiva avviamento motore scambiatore")
      R_Coil( "DB Start motor HYD unit"."Avviamento motore scambiatore"._0 )
   END_RUNG
   RUNG wire#powerrail
      I_Contact( "DB PLC"."Test cesoia"."Disabilitazione motori HYD" )
      I_Contact( "DB Operation mode".Interfaccia.Uscita."Autoreset all'accensione" )
      I_Contact( "DB Operation mode".Interfaccia.Uscita."Comando spegnimento motori" )
      Not()
   END_RUNG wire#w1
   // the same network as SCL:
   IF NOT ("DB Operation mode".Interfaccia.Uscita."Ausiliari inseriti" AND "DB Input cutting-line".Pulsantiere."Pulsantiera principale"."Centralina HYD"."IC Pulsante centralina OFF" AND "DB Start motor HYD unit"."Memorie logiche"."Consenso ciclo avviamento motore scambiatore") OR NOT (NOT "DB PLC"."Test cesoia"."Disabilitazione motori HYD" AND NOT "DB Operation mode".Interfaccia.Uscita."Autoreset all'accensione" AND NOT "DB Operation mode".Interfaccia.Uscita."Comando spegnimento motori") THEN
       "DB Start motor HYD unit"."Memorie logiche"."Fase attiva avviamento motore scambiatore" := 0;
       "DB Start motor HYD unit"."Avviamento motore scambiatore"._0 := FALSE;
   END_IF;
END_REGION

REGION Network 35: Ciclo attivo
   RUNG wire#powerrail
      Contact( "DB Start motor HYD unit"."Memorie logiche"."Consenso ciclo avviamento motore scambiatore" )
      Coil( "DB Start motor HYD unit"."Memorie logiche"."Ciclo attivo motore scambiatore" )
   END_RUNG
   // the same network as SCL:
   "DB Start motor HYD unit"."Memorie logiche"."Ciclo attivo motore scambiatore" := "DB Start motor HYD unit"."Memorie logiche"."Consenso ciclo avviamento motore scambiatore";
END_REGION

REGION Network 36: Inizio ciclo
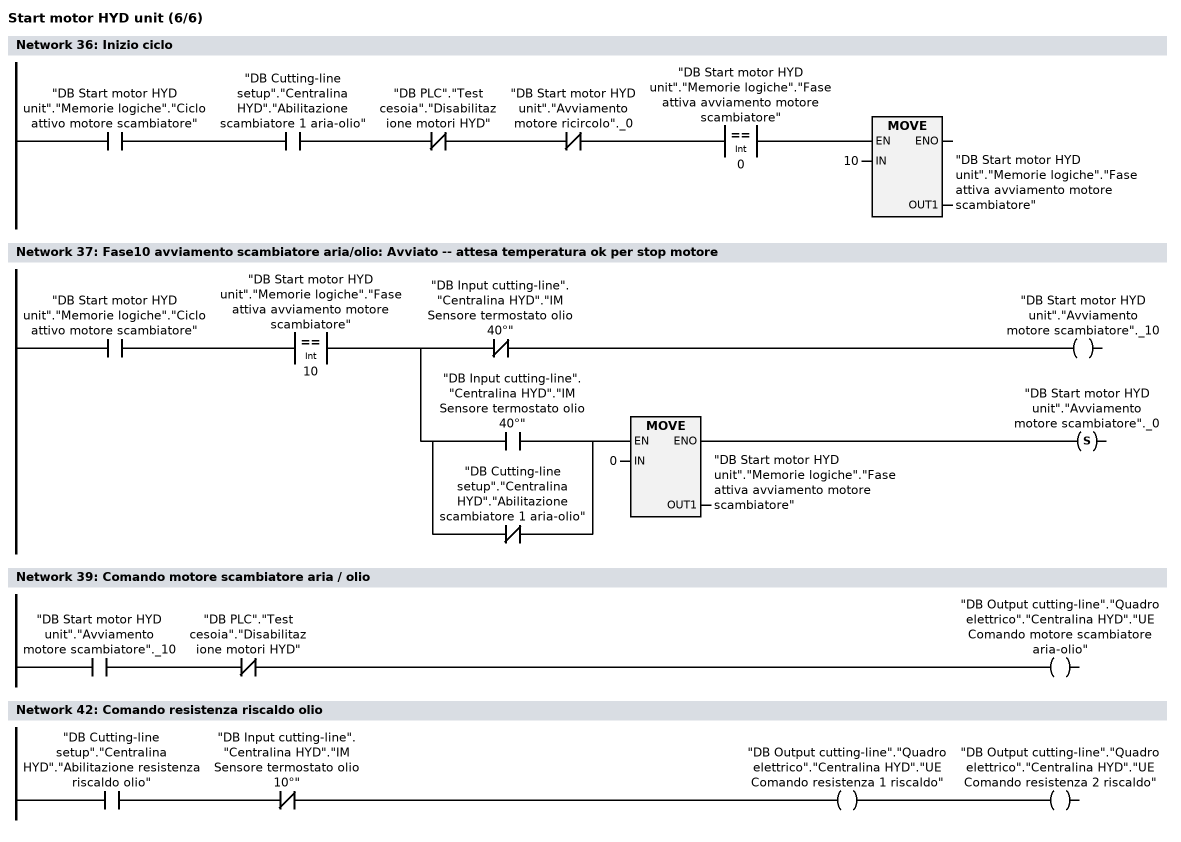
   RUNG wire#powerrail
      Contact( "DB Start motor HYD unit"."Memorie logiche"."Ciclo attivo motore scambiatore" )
      Contact( "DB Cutting-line setup"."Centralina HYD"."Abilitazione scambiatore 1 aria-olio" )
      I_Contact( "DB PLC"."Test cesoia"."Disabilitazione motori HYD" )
      I_Contact( "DB Start motor HYD unit"."Avviamento motore ricircolo"._0 )
      { S7_Templates := "SrcType := Int" } EQ_Contact(in1 := "DB Start motor HYD unit"."Memorie logiche"."Fase attiva avviamento motore scambiatore", in2 := 0)
      Move(in := 10, out1 => "DB Start motor HYD unit"."Memorie logiche"."Fase attiva avviamento motore scambiatore")
   END_RUNG
   // the same network as SCL:
   IF "DB Start motor HYD unit"."Memorie logiche"."Ciclo attivo motore scambiatore" AND "DB Cutting-line setup"."Centralina HYD"."Abilitazione scambiatore 1 aria-olio" AND NOT "DB PLC"."Test cesoia"."Disabilitazione motori HYD" AND NOT "DB Start motor HYD unit"."Avviamento motore ricircolo"._0 AND ("DB Start motor HYD unit"."Memorie logiche"."Fase attiva avviamento motore scambiatore" = 0) THEN
       "DB Start motor HYD unit"."Memorie logiche"."Fase attiva avviamento motore scambiatore" := 10;
   END_IF;
END_REGION

REGION Network 37: Fase10 avviamento scambiatore aria/olio: Avviato -- attesa temperatura ok per stop motore
   RUNG wire#powerrail
      Contact( "DB Start motor HYD unit"."Memorie logiche"."Ciclo attivo motore scambiatore" )
      { S7_Templates := "SrcType := Int" } EQ_Contact(in1 := "DB Start motor HYD unit"."Memorie logiche"."Fase attiva avviamento motore scambiatore", in2 := 10)
      wire#w1
      I_Contact( "DB Input cutting-line"."Centralina HYD"."IM Sensore termostato olio 40°" )
      Coil( "DB Start motor HYD unit"."Avviamento motore scambiatore"._10 )
   END_RUNG
   RUNG wire#w1
      Contact( "DB Input cutting-line"."Centralina HYD"."IM Sensore termostato olio 40°" )
      wire#w2
      Move(in := 0, out1 => "DB Start motor HYD unit"."Memorie logiche"."Fase attiva avviamento motore scambiatore")
      S_Coil( "DB Start motor HYD unit"."Avviamento motore scambiatore"._0 )
   END_RUNG
   RUNG wire#w1
      I_Contact( "DB Cutting-line setup"."Centralina HYD"."Abilitazione scambiatore 1 aria-olio" )
   END_RUNG wire#w2
   // the same network as SCL:
   #_w1 := "DB Start motor HYD unit"."Memorie logiche"."Ciclo attivo motore scambiatore" AND ("DB Start motor HYD unit"."Memorie logiche"."Fase attiva avviamento motore scambiatore" = 10);
   "DB Start motor HYD unit"."Avviamento motore scambiatore"._10 := #_w1 AND NOT "DB Input cutting-line"."Centralina HYD"."IM Sensore termostato olio 40°";
   IF #_w1 AND ("DB Input cutting-line"."Centralina HYD"."IM Sensore termostato olio 40°" OR NOT "DB Cutting-line setup"."Centralina HYD"."Abilitazione scambiatore 1 aria-olio") THEN
       "DB Start motor HYD unit"."Memorie logiche"."Fase attiva avviamento motore scambiatore" := 0;
       "DB Start motor HYD unit"."Avviamento motore scambiatore"._0 := TRUE;
   END_IF;
END_REGION

REGION Network 38: Dummy
END_REGION

REGION Network 39: Comando motore scambiatore aria / olio
   RUNG wire#powerrail
      Contact( "DB Start motor HYD unit"."Avviamento motore scambiatore"._10 )
      I_Contact( "DB PLC"."Test cesoia"."Disabilitazione motori HYD" )
      Coil( "DB Output cutting-line"."Quadro elettrico"."Centralina HYD"."UE Comando motore scambiatore aria-olio" )
   END_RUNG
   // the same network as SCL:
   "DB Output cutting-line"."Quadro elettrico"."Centralina HYD"."UE Comando motore scambiatore aria-olio" := "DB Start motor HYD unit"."Avviamento motore scambiatore"._10 AND NOT "DB PLC"."Test cesoia"."Disabilitazione motori HYD";
END_REGION

REGION Network 40: Dummy
END_REGION

REGION Network 41: ****************************** Resistenza di riscaldo ***********************************
END_REGION

REGION Network 42: Comando resistenza riscaldo olio
   RUNG wire#powerrail
      Contact( "DB Cutting-line setup"."Centralina HYD"."Abilitazione resistenza riscaldo olio" )
      I_Contact( "DB Input cutting-line"."Centralina HYD"."IM Sensore termostato olio 10°" )
      Coil( "DB Output cutting-line"."Quadro elettrico"."Centralina HYD"."UE Comando resistenza 1 riscaldo" )
      Coil( "DB Output cutting-line"."Quadro elettrico"."Centralina HYD"."UE Comando resistenza 2 riscaldo" )
   END_RUNG
   // the same network as SCL:
   "DB Output cutting-line"."Quadro elettrico"."Centralina HYD"."UE Comando resistenza 1 riscaldo" := "DB Cutting-line setup"."Centralina HYD"."Abilitazione resistenza riscaldo olio" AND NOT "DB Input cutting-line"."Centralina HYD"."IM Sensore termostato olio 10°";
   "DB Output cutting-line"."Quadro elettrico"."Centralina HYD"."UE Comando resistenza 2 riscaldo" := "DB Output cutting-line"."Quadro elettrico"."Centralina HYD"."UE Comando resistenza 1 riscaldo";
END_REGION

REGION Network 43: Dummy
END_REGION
END_FUNCTION
